TYPE ST_BASE_SETTINGS :
STRUCT
	name:			T_SHORT_STR := IING.STRING_BASE_SETTINGS_INITIAL_NAME;
	doHide:			BOOL := TRUE;
END_STRUCT
END_TYPE

(* stored: Version 1.1.0.1, ProductVersion 3.1.4026.18
   DUT ST_BASE_SETTINGS: Id {cc54904e-32c4-4396-bb92-faebd69be2db} *)
